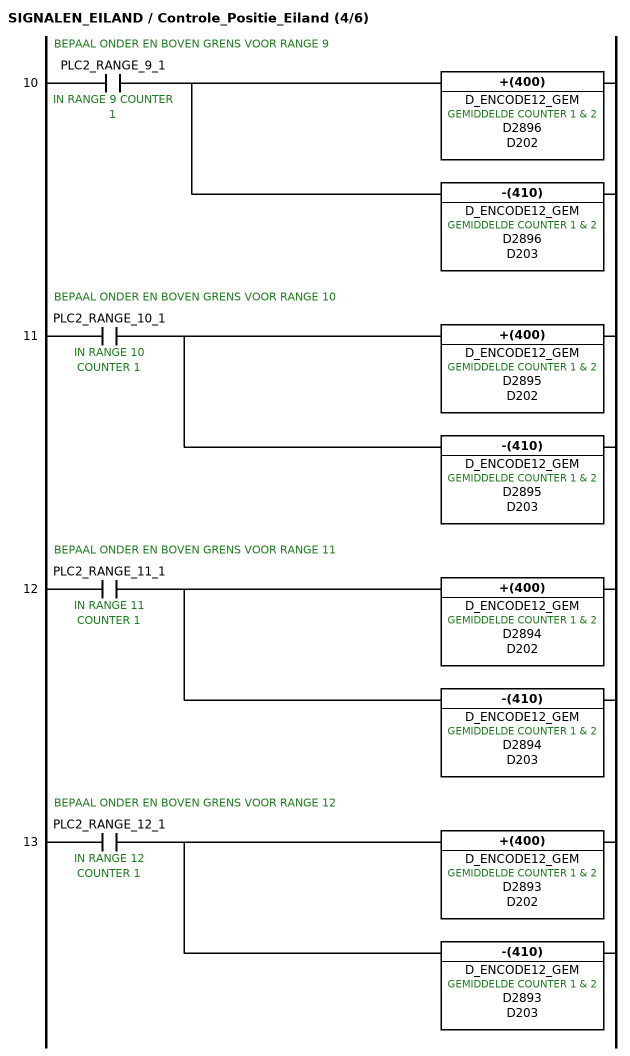
; [picture p397: SIGNALEN_EILAND / Controle_Positie_Eiland, rungs 10-13]
; rung 10: BEPAAL ONDER EN BOVEN GRENS VOOR RANGE 9
LD PLC2_RANGE_9_1  ; IN RANGE 9 COUNTER 1
+(400) D_ENCODE12_GEM D2896 D202  ; GEMIDDELDE COUNTER 1 & 2
-(410) D_ENCODE12_GEM D2896 D203  ; GEMIDDELDE COUNTER 1 & 2
; rung 11: BEPAAL ONDER EN BOVEN GRENS VOOR RANGE 10
LD PLC2_RANGE_10_1  ; IN RANGE 10 COUNTER 1
+(400) D_ENCODE12_GEM D2895 D202  ; GEMIDDELDE COUNTER 1 & 2
-(410) D_ENCODE12_GEM D2895 D203  ; GEMIDDELDE COUNTER 1 & 2
; rung 12: BEPAAL ONDER EN BOVEN GRENS VOOR RANGE 11
LD PLC2_RANGE_11_1  ; IN RANGE 11 COUNTER 1
+(400) D_ENCODE12_GEM D2894 D202  ; GEMIDDELDE COUNTER 1 & 2
-(410) D_ENCODE12_GEM D2894 D203  ; GEMIDDELDE COUNTER 1 & 2
; rung 13: BEPAAL ONDER EN BOVEN GRENS VOOR RANGE 12
LD PLC2_RANGE_12_1  ; IN RANGE 12 COUNTER 1
+(400) D_ENCODE12_GEM D2893 D202  ; GEMIDDELDE COUNTER 1 & 2
-(410) D_ENCODE12_GEM D2893 D203  ; GEMIDDELDE COUNTER 1 & 2

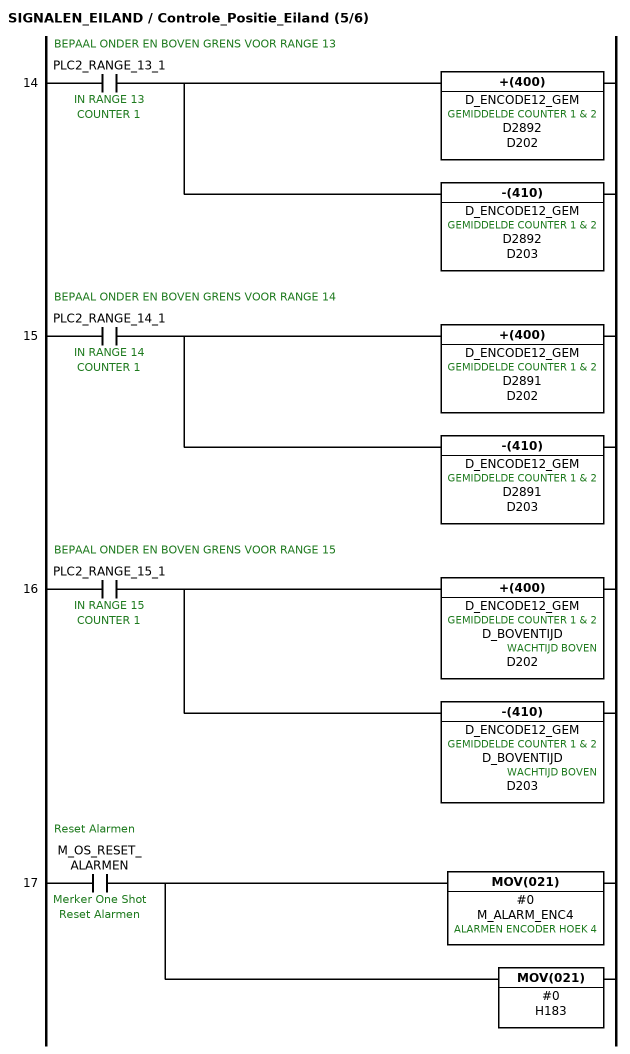
; rung 14: BEPAAL ONDER EN BOVEN GRENS VOOR RANGE 13
LD PLC2_RANGE_13_1  ; IN RANGE 13 COUNTER 1
+(400) D_ENCODE12_GEM D2892 D202  ; GEMIDDELDE COUNTER 1 & 2
-(410) D_ENCODE12_GEM D2892 D203  ; GEMIDDELDE COUNTER 1 & 2
; rung 15: BEPAAL ONDER EN BOVEN GRENS VOOR RANGE 14
LD PLC2_RANGE_14_1  ; IN RANGE 14 COUNTER 1
+(400) D_ENCODE12_GEM D2891 D202  ; GEMIDDELDE COUNTER 1 & 2
-(410) D_ENCODE12_GEM D2891 D203  ; GEMIDDELDE COUNTER 1 & 2
; rung 16: BEPAAL ONDER EN BOVEN GRENS VOOR RANGE 15
LD PLC2_RANGE_15_1  ; IN RANGE 15 COUNTER 1
+(400) D_ENCODE12_GEM D_BOVENTIJD D202  ; GEMIDDELDE COUNTER 1 & 2, WACHTIJD BOVEN
-(410) D_ENCODE12_GEM D_BOVENTIJD D203  ; GEMIDDELDE COUNTER 1 & 2, WACHTIJD BOVEN
; rung 17: Reset Alarmen
LD M_OS_RESET_ALARMEN  ; Merker One Shot Reset Alarmen
MOV(021) #0 M_ALARM_ENC4  ; ALARMEN ENCODER HOEK 4
MOV(021) #0 H183

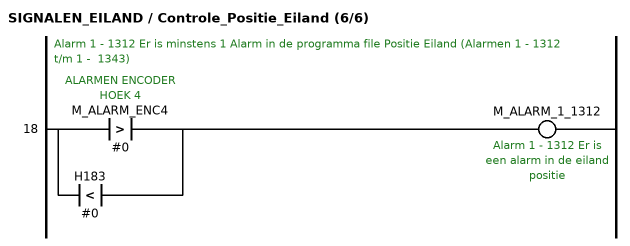
; rung 18: Alarm 1 - 1312 Er is minstens 1 Alarm in de programma file Positie Eiland (Alarmen 1 - 1312 t/m 1 -  1343)
LD>(320) M_ALARM_ENC4 #0  ; ALARMEN ENCODER HOEK 4
OR<(310) H183 #0
OUT M_ALARM_1_1312  ; Alarm 1 - 1312 Er is een alarm in de eiland positie

### Section Controle_Level_Switches_Eiland

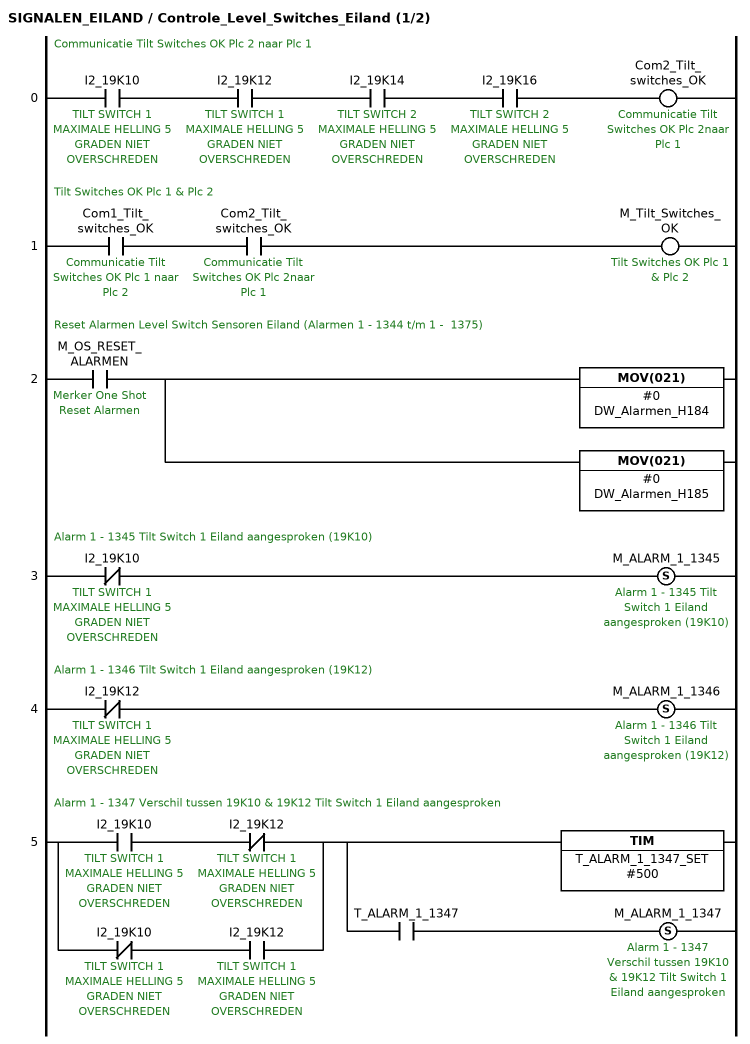
; rung 0: Communicatie Tilt Switches OK Plc 2 naar Plc 1
LD I2_19K10  ; TILT SWITCH 1 MAXIMALE HELLING 5 GRADEN NIET OVERSCHREDEN
AND I2_19K12  ; TILT SWITCH 1 MAXIMALE HELLING 5 GRADEN NIET OVERSCHREDEN
AND I2_19K14  ; TILT SWITCH 2 MAXIMALE HELLING 5 GRADEN NIET OVERSCHREDEN
AND I2_19K16  ; TILT SWITCH 2 MAXIMALE HELLING 5 GRADEN NIET OVERSCHREDEN
OUT Com2_Tilt_switches_OK  ; Communicatie Tilt Switches OK Plc 2naar Plc 1
; rung 1: Tilt Switches OK Plc 1 & Plc 2
LD Com1_Tilt_switches_OK  ; Communicatie Tilt Switches OK Plc 1 naar Plc 2
AND Com2_Tilt_switches_OK  ; Communicatie Tilt Switches OK Plc 2naar Plc 1
OUT M_Tilt_Switches_OK  ; Tilt Switches OK Plc 1 & Plc 2
; rung 2: Reset Alarmen Level Switch Sensoren Eiland (Alarmen 1 - 1344 t/m 1 -  1375)
LD M_OS_RESET_ALARMEN  ; Merker One Shot Reset Alarmen
MOV(021) #0 DW_Alarmen_H184
MOV(021) #0 DW_Alarmen_H185
; rung 3: Alarm 1 - 1345 Tilt Switch 1 Eiland aangesproken (19K10)
LDNOT I2_19K10  ; TILT SWITCH 1 MAXIMALE HELLING 5 GRADEN NIET OVERSCHREDEN
SET M_ALARM_1_1345  ; Alarm 1 - 1345 Tilt Switch 1 Eiland aangesproken (19K10)
; rung 4: Alarm 1 - 1346 Tilt Switch 1 Eiland aangesproken (19K12)
LDNOT I2_19K12  ; TILT SWITCH 1 MAXIMALE HELLING 5 GRADEN NIET OVERSCHREDEN
SET M_ALARM_1_1346  ; Alarm 1 - 1346 Tilt Switch 1 Eiland aangesproken (19K12)
; rung 5: Alarm 1 - 1347 Verschil tussen 19K10 & 19K12 Tilt Switch 1 Eiland aangesproken
LD I2_19K10  ; TILT SWITCH 1 MAXIMALE HELLING 5 GRADEN NIET OVERSCHREDEN
ANDNOT I2_19K12  ; TILT SWITCH 1 MAXIMALE HELLING 5 GRADEN NIET OVERSCHREDEN
LDNOT I2_19K10  ; TILT SWITCH 1 MAXIMALE HELLING 5 GRADEN NIET OVERSCHREDEN
AND I2_19K12  ; TILT SWITCH 1 MAXIMALE HELLING 5 GRADEN NIET OVERSCHREDEN
ORLD
TIM T_ALARM_1_1347_SET #500
AND T_ALARM_1_1347
SET M_ALARM_1_1347  ; Alarm 1 - 1347 Verschil tussen 19K10 & 19K12 Tilt Switch 1 Eiland aangesproken

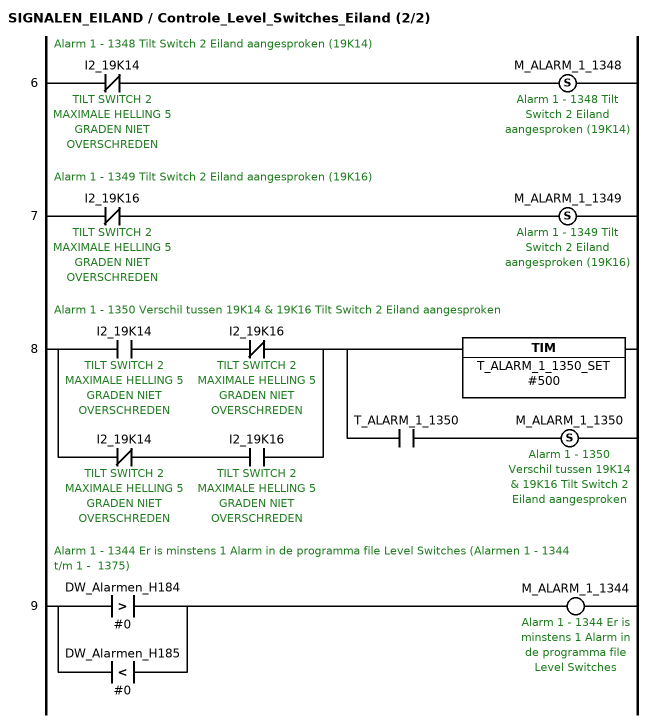
; rung 6: Alarm 1 - 1348 Tilt Switch 2 Eiland aangesproken (19K14)
LDNOT I2_19K14  ; TILT SWITCH 2 MAXIMALE HELLING 5 GRADEN NIET OVERSCHREDEN
SET M_ALARM_1_1348  ; Alarm 1 - 1348 Tilt Switch 2 Eiland aangesproken (19K14)
; rung 7: Alarm 1 - 1349 Tilt Switch 2 Eiland aangesproken (19K16)
LDNOT I2_19K16  ; TILT SWITCH 2 MAXIMALE HELLING 5 GRADEN NIET OVERSCHREDEN
SET M_ALARM_1_1349  ; Alarm 1 - 1349 Tilt Switch 2 Eiland aangesproken (19K16)
; rung 8: Alarm 1 - 1350 Verschil tussen 19K14 & 19K16 Tilt Switch 2 Eiland aangesproken
LD I2_19K14  ; TILT SWITCH 2 MAXIMALE HELLING 5 GRADEN NIET OVERSCHREDEN
ANDNOT I2_19K16  ; TILT SWITCH 2 MAXIMALE HELLING 5 GRADEN NIET OVERSCHREDEN
LDNOT I2_19K14  ; TILT SWITCH 2 MAXIMALE HELLING 5 GRADEN NIET OVERSCHREDEN
AND I2_19K16  ; TILT SWITCH 2 MAXIMALE HELLING 5 GRADEN NIET OVERSCHREDEN
ORLD
TIM T_ALARM_1_1350_SET #500
AND T_ALARM_1_1350
SET M_ALARM_1_1350  ; Alarm 1 - 1350 Verschil tussen 19K14 & 19K16 Tilt Switch 2 Eiland aangesproken
; rung 9: Alarm 1 - 1344 Er is minstens 1 Alarm in de programma file Level Switches (Alarmen 1 - 1344 t/m 1 -  1375)
LD>(320) DW_Alarmen_H184 #0
OR<(310) DW_Alarmen_H185 #0
OUT M_ALARM_1_1344  ; Alarm 1 - 1344 Er is minstens 1 Alarm in de programma file Level Switches

### Section Einde_Signalering_Eiland
; rung 0
END(001)

## Program BESTURING_EILAND (cyclic task 11)
Local symbols
Com1_Eiland_Rond_Geweest 3047.14 BOOL
Com1_Hydrauliek_Eiland_Inbedrijf 3045.15 BOOL
Com2_Eiland_Rond_Geweest 3347.14 BOOL
Com2_Hydrauliek_Eiland_Inbedrijf 3345.15 BOOL
M_ALARM_2_1515 H194.11 BOOL  ; Alarm 2 - 1515 Thermistor Fout Motor 2 Eiland (13R7 / 13U6 / 13K9)
M_Hoofdpomp_Hydrau_Eiland W220.03 BOOL  ; Start Hoofdpomp Hydrauliek Eiland

### Section Poortjes_Eiland

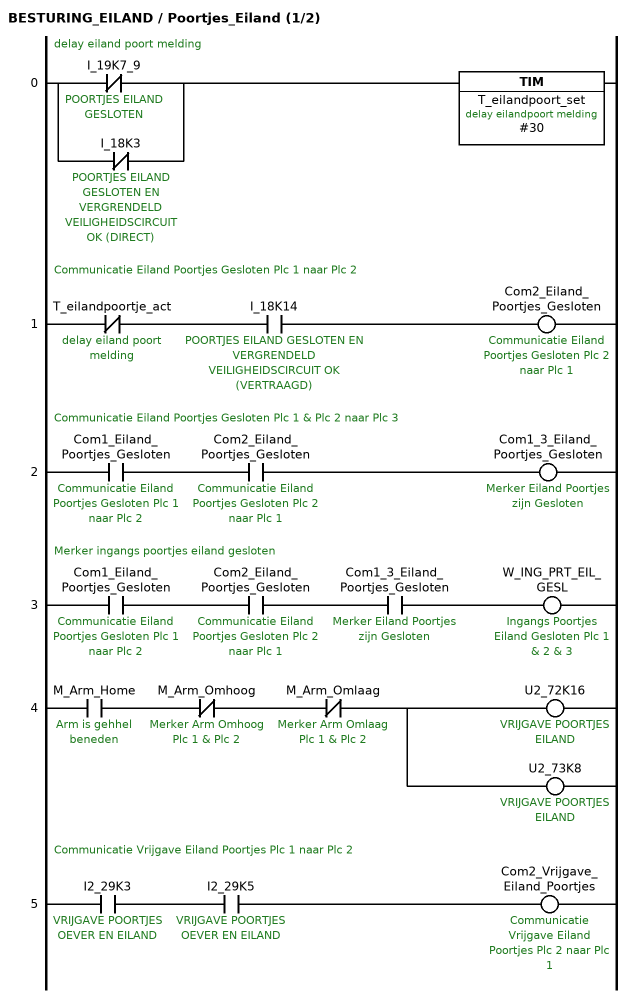
; rung 0: delay eiland poort melding
LDNOT I_19K7_9  ; POORTJES EILAND GESLOTEN
ORNOT I_18K3  ; POORTJES EILAND GESLOTEN EN VERGRENDELD VEILIGHEIDSCIRCUIT OK (DIRECT)
TIM T_eilandpoort_set #30  ; delay eilandpoort melding
; rung 1: Communicatie Eiland Poortjes Gesloten Plc 1 naar Plc 2
LDNOT T_eilandpoortje_act  ; delay eiland poort melding
AND I_18K14  ; POORTJES EILAND GESLOTEN EN VERGRENDELD VEILIGHEIDSCIRCUIT OK (VERTRAAGD)
OUT Com2_Eiland_Poortjes_Gesloten  ; Communicatie Eiland Poortjes Gesloten Plc 2 naar Plc 1
; rung 2: Communicatie Eiland Poortjes Gesloten Plc 1 & Plc 2 naar Plc 3
LD Com1_Eiland_Poortjes_Gesloten  ; Communicatie Eiland Poortjes Gesloten Plc 1 naar Plc 2
AND Com2_Eiland_Poortjes_Gesloten  ; Communicatie Eiland Poortjes Gesloten Plc 2 naar Plc 1
OUT Com1_3_Eiland_Poortjes_Gesloten  ; Merker Eiland Poortjes zijn Gesloten
; rung 3: Merker ingangs poortjes eiland gesloten
LD Com1_Eiland_Poortjes_Gesloten  ; Communicatie Eiland Poortjes Gesloten Plc 1 naar Plc 2
AND Com2_Eiland_Poortjes_Gesloten  ; Communicatie Eiland Poortjes Gesloten Plc 2 naar Plc 1
AND Com1_3_Eiland_Poortjes_Gesloten  ; Merker Eiland Poortjes zijn Gesloten
OUT W_ING_PRT_EIL_GESL  ; Ingangs Poortjes Eiland Gesloten Plc 1 & 2 & 3
; rung 4
LD M_Arm_Home  ; Arm is gehhel beneden
ANDNOT M_Arm_Omhoog  ; Merker Arm Omhoog Plc 1 & Plc 2
ANDNOT M_Arm_Omlaag  ; Merker Arm Omlaag Plc 1 & Plc 2
OUT U2_72K16  ; VRIJGAVE POORTJES EILAND
OUT U2_73K8  ; VRIJGAVE POORTJES EILAND
; rung 5: Communicatie Vrijgave Eiland Poortjes Plc 1 naar Plc 2
LD I2_29K3  ; VRIJGAVE POORTJES OEVER EN EILAND
AND I2_29K5  ; VRIJGAVE POORTJES OEVER EN EILAND
OUT Com2_Vrijgave_Eiland_Poortjes  ; Communicatie Vrijgave Eiland Poortjes Plc 2 naar Plc 1

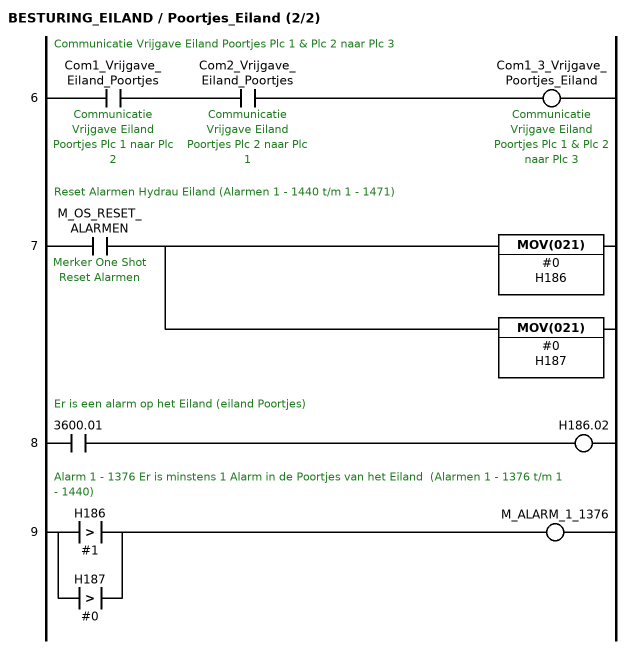
; rung 6: Communicatie Vrijgave Eiland Poortjes Plc 1 & Plc 2 naar Plc 3
LD Com1_Vrijgave_Eiland_Poortjes  ; Communicatie Vrijgave Eiland Poortjes Plc 1 naar Plc 2
AND Com2_Vrijgave_Eiland_Poortjes  ; Communicatie Vrijgave Eiland Poortjes Plc 2 naar Plc 1
OUT Com1_3_Vrijgave_Poortjes_Eiland  ; Communicatie Vrijgave Eiland Poortjes Plc 1 & Plc 2 naar Plc 3
; rung 7: Reset Alarmen Hydrau Eiland (Alarmen 1 - 1440 t/m 1 - 1471)
LD M_OS_RESET_ALARMEN  ; Merker One Shot Reset Alarmen
MOV(021) #0 H186
MOV(021) #0 H187
; rung 8: Er is een alarm op het Eiland (eiland Poortjes)
LD 3600.01
OUT H186.02
; rung 9: Alarm 1 - 1376 Er is minstens 1 Alarm in de Poortjes van het Eiland  (Alarmen 1 - 1376 t/m 1 - 1440)
LD>(320) H186 #1
OR>(320) H187 #0
OUT M_ALARM_1_1376

### Section Hydrauliek_Eiland

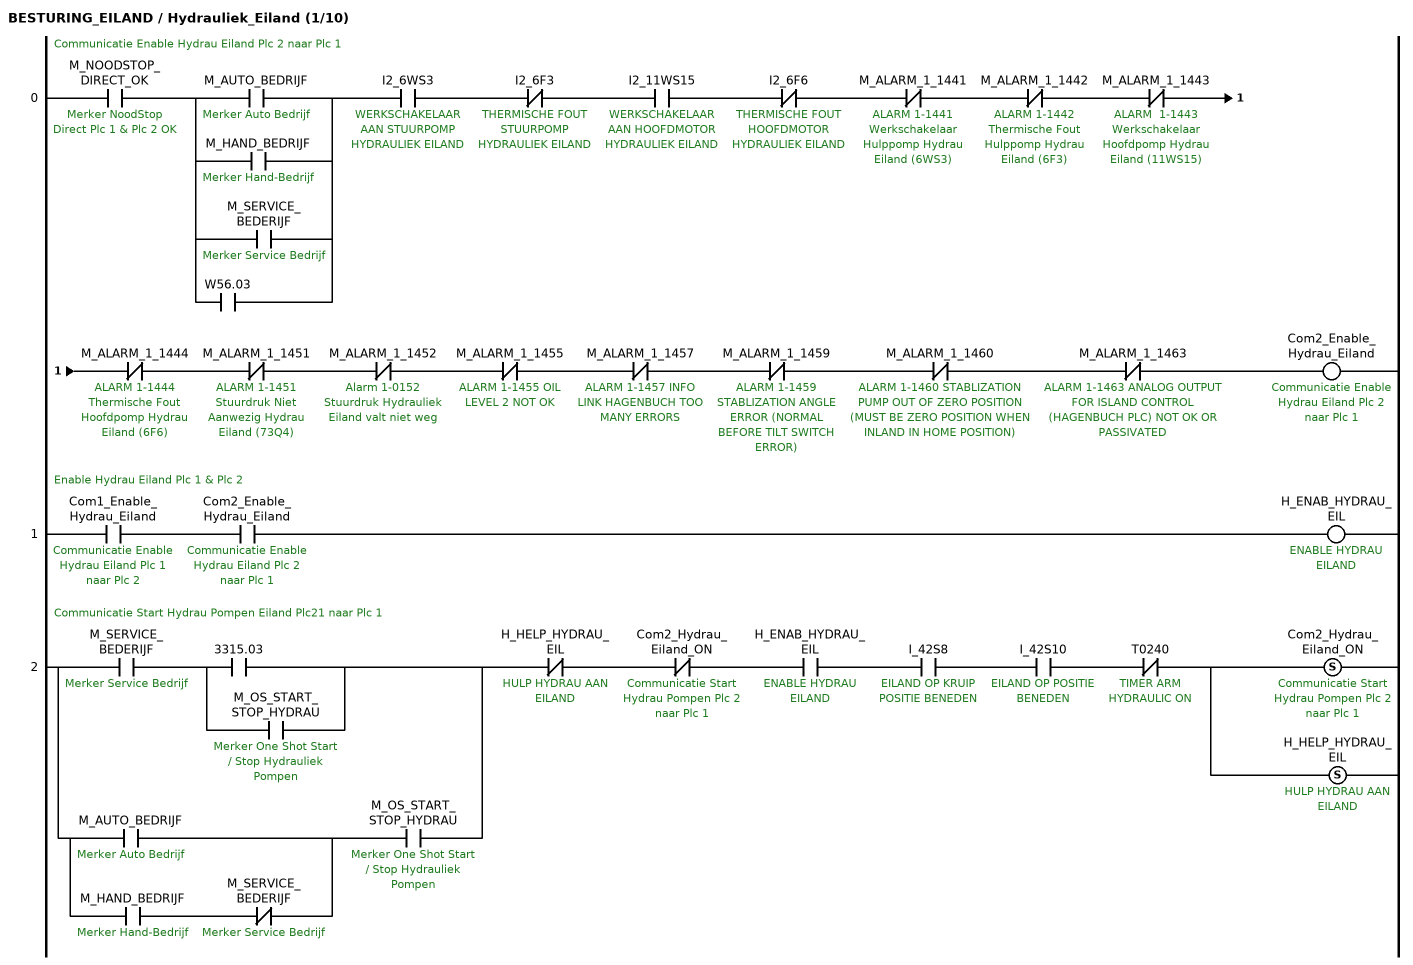
; rung 0: Communicatie Enable Hydrau Eiland Plc 2 naar Plc 1
LD M_NOODSTOP_DIRECT_OK  ; Merker NoodStop Direct Plc 1 & Plc 2 OK
LD M_AUTO_BEDRIJF  ; Merker Auto Bedrijf
OR M_HAND_BEDRIJF  ; Merker Hand-Bedrijf
OR M_SERVICE_BEDERIJF  ; Merker Service Bedrijf
OR W56.03
ANDLD
AND I2_6WS3  ; WERKSCHAKELAAR AAN STUURPOMP HYDRAULIEK EILAND
ANDNOT I2_6F3  ; THERMISCHE FOUT STUURPOMP HYDRAULIEK EILAND
AND I2_11WS15  ; WERKSCHAKELAAR AAN HOOFDMOTOR HYDRAULIEK EILAND
ANDNOT I2_6F6  ; THERMISCHE FOUT HOOFDMOTOR HYDRAULIEK EILAND
ANDNOT M_ALARM_1_1441  ; ALARM 1-1441 Werkschakelaar Hulppomp Hydrau Eiland (6WS3)
ANDNOT M_ALARM_1_1442  ; ALARM 1-1442 Thermische Fout Hulppomp Hydrau Eiland (6F3)
ANDNOT M_ALARM_1_1443  ; ALARM  1-1443 Werkschakelaar Hoofdpomp Hydrau Eiland (11WS15)
ANDNOT M_ALARM_1_1444  ; ALARM 1-1444 Thermische Fout Hoofdpomp Hydrau Eiland (6F6)
ANDNOT M_ALARM_1_1451  ; ALARM 1-1451 Stuurdruk Niet Aanwezig Hydrau Eiland (73Q4)
ANDNOT M_ALARM_1_1452  ; Alarm 1-0152 Stuurdruk Hydrauliek Eiland valt niet weg
ANDNOT M_ALARM_1_1455  ; ALARM 1-1455 OIL LEVEL 2 NOT OK
ANDNOT M_ALARM_1_1457  ; ALARM 1-1457 INFO LINK HAGENBUCH TOO MANY ERRORS
ANDNOT M_ALARM_1_1459  ; ALARM 1-1459 STABLIZATION ANGLE ERROR (NORMAL BEFORE TILT SWITCH ERROR)
ANDNOT M_ALARM_1_1460  ; ALARM 1-1460 STABLIZATION PUMP OUT OF ZERO POSITION (MUST BE ZERO POSITION WHEN INLAND IN HOME POSITION)
ANDNOT M_ALARM_1_1463  ; ALARM 1-1463 ANALOG OUTPUT FOR ISLAND CONTROL (HAGENBUCH PLC) NOT OK OR PASSIVATED
OUT Com2_Enable_Hydrau_Eiland  ; Communicatie Enable Hydrau Eiland Plc 2 naar Plc 1
; rung 1: Enable Hydrau Eiland Plc 1 & Plc 2
LD Com1_Enable_Hydrau_Eiland  ; Communicatie Enable Hydrau Eiland Plc 1 naar Plc 2
AND Com2_Enable_Hydrau_Eiland  ; Communicatie Enable Hydrau Eiland Plc 2 naar Plc 1
OUT H_ENAB_HYDRAU_EIL  ; ENABLE HYDRAU EILAND
; rung 2: Communicatie Start Hydrau Pompen Eiland Plc21 naar Plc 1
LD M_SERVICE_BEDERIJF  ; Merker Service Bedrijf
LD 3315.03
OR M_OS_START_STOP_HYDRAU  ; Merker One Shot Start / Stop Hydrauliek Pompen
ANDLD
LD M_AUTO_BEDRIJF  ; Merker Auto Bedrijf
LD M_HAND_BEDRIJF  ; Merker Hand-Bedrijf
ANDNOT M_SERVICE_BEDERIJF  ; Merker Service Bedrijf
ORLD
AND M_OS_START_STOP_HYDRAU  ; Merker One Shot Start / Stop Hydrauliek Pompen
ORLD
ANDNOT H_HELP_HYDRAU_EIL  ; HULP HYDRAU AAN EILAND
ANDNOT Com2_Hydrau_Eiland_ON  ; Communicatie Start Hydrau Pompen Plc 2 naar Plc 1
AND H_ENAB_HYDRAU_EIL  ; ENABLE HYDRAU EILAND
AND I_42S8  ; EILAND OP KRUIP POSITIE BENEDEN
AND I_42S10  ; EILAND OP POSITIE BENEDEN
ANDNOT T0240  ; TIMER ARM HYDRAULIC ON
SET Com2_Hydrau_Eiland_ON  ; Communicatie Start Hydrau Pompen Plc 2 naar Plc 1
SET H_HELP_HYDRAU_EIL  ; HULP HYDRAU AAN EILAND

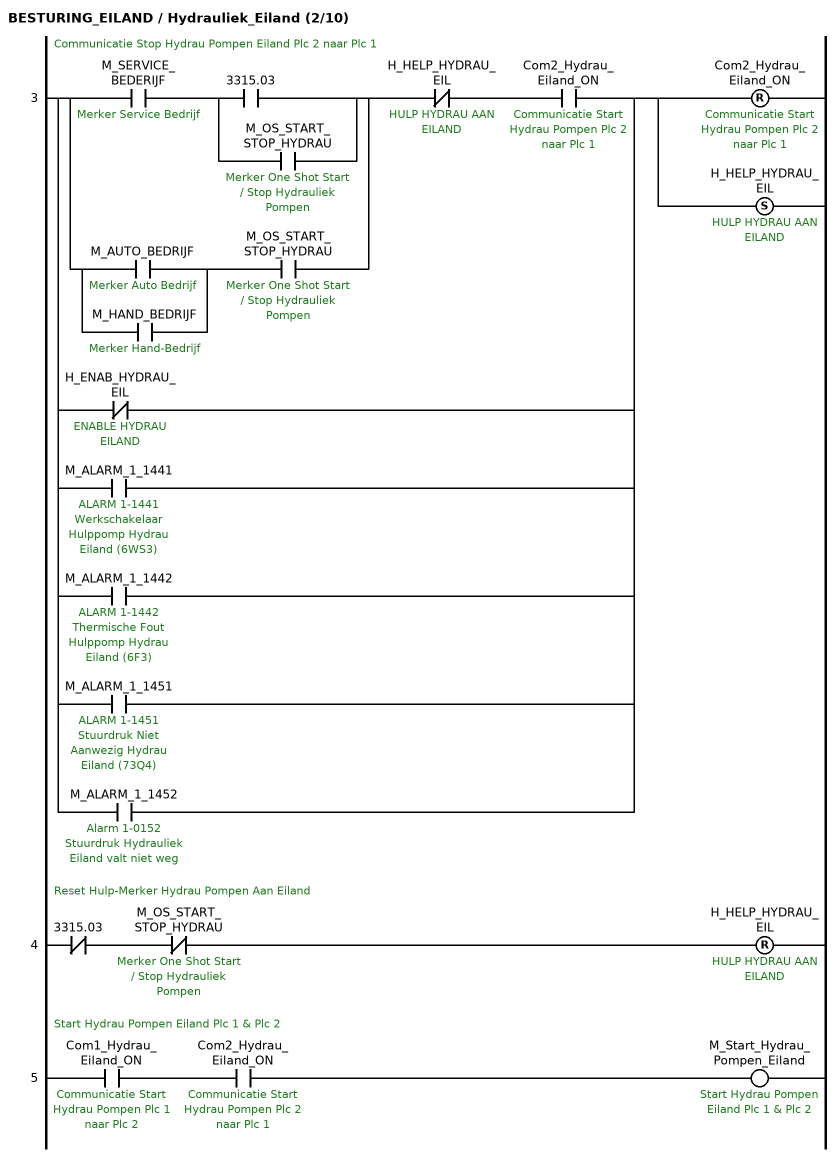
; rung 3: Communicatie Stop Hydrau Pompen Eiland Plc 2 naar Plc 1
LD M_SERVICE_BEDERIJF  ; Merker Service Bedrijf
LD 3315.03
OR M_OS_START_STOP_HYDRAU  ; Merker One Shot Start / Stop Hydrauliek Pompen
ANDLD
LD M_AUTO_BEDRIJF  ; Merker Auto Bedrijf
OR M_HAND_BEDRIJF  ; Merker Hand-Bedrijf
AND M_OS_START_STOP_HYDRAU  ; Merker One Shot Start / Stop Hydrauliek Pompen
ORLD
ANDNOT H_HELP_HYDRAU_EIL  ; HULP HYDRAU AAN EILAND
AND Com2_Hydrau_Eiland_ON  ; Communicatie Start Hydrau Pompen Plc 2 naar Plc 1
ORNOT H_ENAB_HYDRAU_EIL  ; ENABLE HYDRAU EILAND
OR M_ALARM_1_1441  ; ALARM 1-1441 Werkschakelaar Hulppomp Hydrau Eiland (6WS3)
OR M_ALARM_1_1442  ; ALARM 1-1442 Thermische Fout Hulppomp Hydrau Eiland (6F3)
OR M_ALARM_1_1451  ; ALARM 1-1451 Stuurdruk Niet Aanwezig Hydrau Eiland (73Q4)
OR M_ALARM_1_1452  ; Alarm 1-0152 Stuurdruk Hydrauliek Eiland valt niet weg
RSET Com2_Hydrau_Eiland_ON  ; Communicatie Start Hydrau Pompen Plc 2 naar Plc 1
SET H_HELP_HYDRAU_EIL  ; HULP HYDRAU AAN EILAND
; rung 4: Reset Hulp-Merker Hydrau Pompen Aan Eiland
LDNOT 3315.03
ANDNOT M_OS_START_STOP_HYDRAU  ; Merker One Shot Start / Stop Hydrauliek Pompen
RSET H_HELP_HYDRAU_EIL  ; HULP HYDRAU AAN EILAND
; rung 5: Start Hydrau Pompen Eiland Plc 1 & Plc 2
LD Com1_Hydrau_Eiland_ON  ; Communicatie Start Hydrau Pompen Plc 1 naar Plc 2
AND Com2_Hydrau_Eiland_ON  ; Communicatie Start Hydrau Pompen Plc 2 naar Plc 1
OUT M_Start_Hydrau_Pompen_Eiland  ; Start Hydrau Pompen Eiland Plc 1 & Plc 2

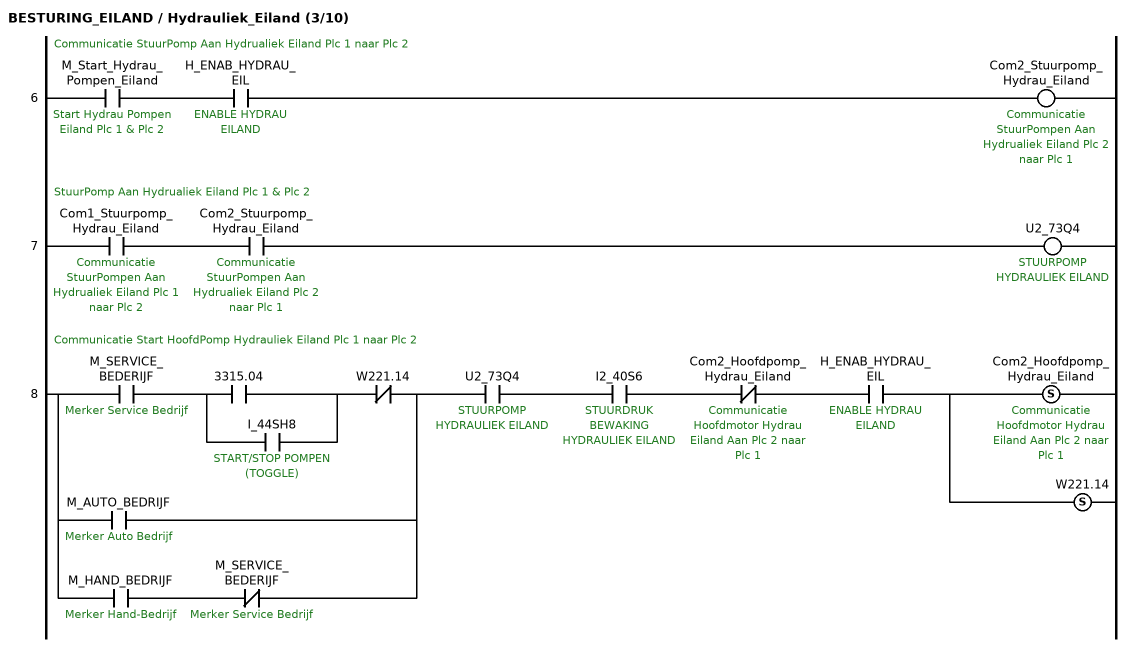
; rung 6: Communicatie StuurPomp Aan Hydrualiek Eiland Plc 1 naar Plc 2
LD M_Start_Hydrau_Pompen_Eiland  ; Start Hydrau Pompen Eiland Plc 1 & Plc 2
AND H_ENAB_HYDRAU_EIL  ; ENABLE HYDRAU EILAND
OUT Com2_Stuurpomp_Hydrau_Eiland  ; Communicatie StuurPompen Aan Hydrualiek Eiland Plc 2 naar Plc 1
; rung 7: StuurPomp Aan Hydrualiek Eiland Plc 1 & Plc 2
LD Com1_Stuurpomp_Hydrau_Eiland  ; Communicatie StuurPompen Aan Hydrualiek Eiland Plc 1 naar Plc 2
AND Com2_Stuurpomp_Hydrau_Eiland  ; Communicatie StuurPompen Aan Hydrualiek Eiland Plc 2 naar Plc 1
OUT U2_73Q4  ; STUURPOMP HYDRAULIEK EILAND
; rung 8: Communicatie Start HoofdPomp Hydrauliek Eiland Plc 1 naar Plc 2
LD M_SERVICE_BEDERIJF  ; Merker Service Bedrijf
LD 3315.04
OR I_44SH8  ; START/STOP POMPEN (TOGGLE)
ANDLD
ANDNOT W221.14
OR M_AUTO_BEDRIJF  ; Merker Auto Bedrijf
LD M_HAND_BEDRIJF  ; Merker Hand-Bedrijf
ANDNOT M_SERVICE_BEDERIJF  ; Merker Service Bedrijf
ORLD
AND U2_73Q4  ; STUURPOMP HYDRAULIEK EILAND
AND I2_40S6  ; STUURDRUK BEWAKING HYDRAULIEK EILAND
ANDNOT Com2_Hoofdpomp_Hydrau_Eiland  ; Communicatie Hoofdmotor Hydrau Eiland Aan Plc 2 naar Plc 1
AND H_ENAB_HYDRAU_EIL  ; ENABLE HYDRAU EILAND
SET Com2_Hoofdpomp_Hydrau_Eiland  ; Communicatie Hoofdmotor Hydrau Eiland Aan Plc 2 naar Plc 1
SET W221.14

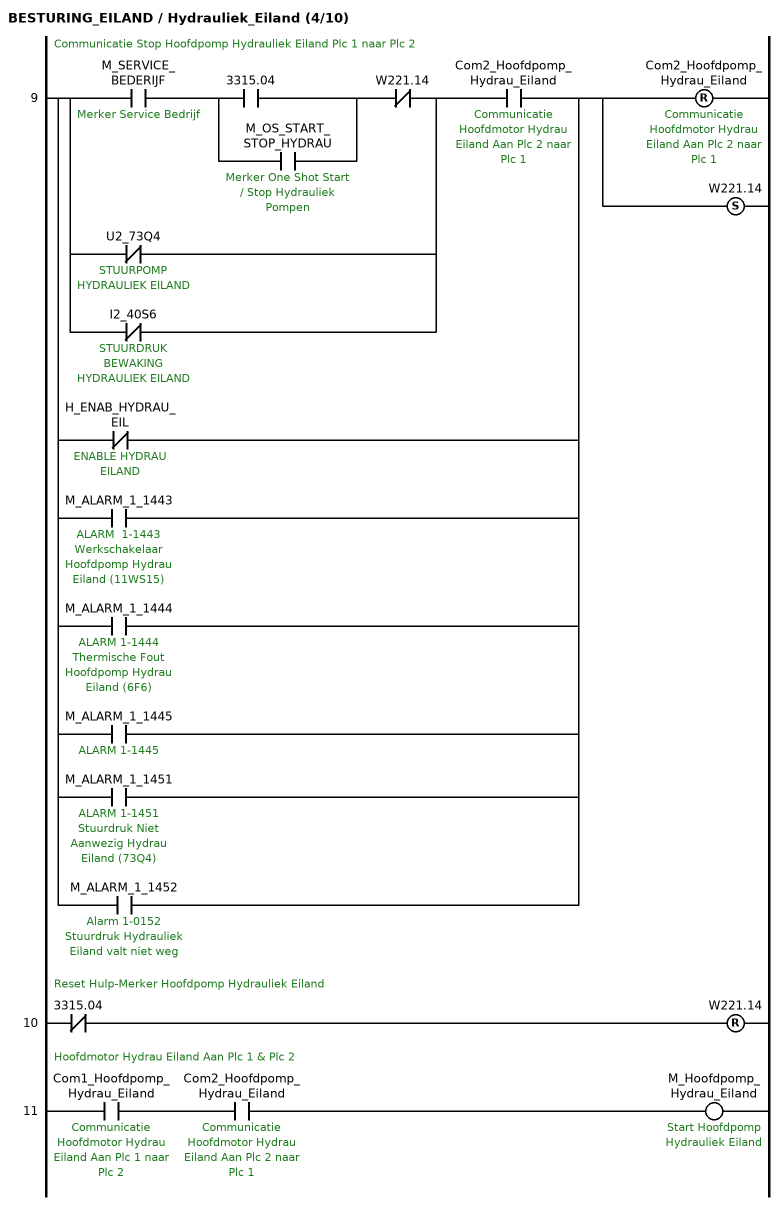
; rung 9: Communicatie Stop Hoofdpomp Hydrauliek Eiland Plc 1 naar Plc 2
LD M_SERVICE_BEDERIJF  ; Merker Service Bedrijf
LD 3315.04
OR M_OS_START_STOP_HYDRAU  ; Merker One Shot Start / Stop Hydrauliek Pompen
ANDLD
ANDNOT W221.14
ORNOT U2_73Q4  ; STUURPOMP HYDRAULIEK EILAND
ORNOT I2_40S6  ; STUURDRUK BEWAKING HYDRAULIEK EILAND
AND Com2_Hoofdpomp_Hydrau_Eiland  ; Communicatie Hoofdmotor Hydrau Eiland Aan Plc 2 naar Plc 1
ORNOT H_ENAB_HYDRAU_EIL  ; ENABLE HYDRAU EILAND
OR M_ALARM_1_1443  ; ALARM  1-1443 Werkschakelaar Hoofdpomp Hydrau Eiland (11WS15)
OR M_ALARM_1_1444  ; ALARM 1-1444 Thermische Fout Hoofdpomp Hydrau Eiland (6F6)
OR M_ALARM_1_1445  ; ALARM 1-1445
OR M_ALARM_1_1451  ; ALARM 1-1451 Stuurdruk Niet Aanwezig Hydrau Eiland (73Q4)
OR M_ALARM_1_1452  ; Alarm 1-0152 Stuurdruk Hydrauliek Eiland valt niet weg
RSET Com2_Hoofdpomp_Hydrau_Eiland  ; Communicatie Hoofdmotor Hydrau Eiland Aan Plc 2 naar Plc 1
SET W221.14
; rung 10: Reset Hulp-Merker Hoofdpomp Hydrauliek Eiland
LDNOT 3315.04
RSET W221.14
; rung 11: Hoofdmotor Hydrau Eiland Aan Plc 1 & Plc 2
LD Com1_Hoofdpomp_Hydrau_Eiland  ; Communicatie Hoofdmotor Hydrau Eiland Aan Plc 1 naar Plc 2
AND Com2_Hoofdpomp_Hydrau_Eiland  ; Communicatie Hoofdmotor Hydrau Eiland Aan Plc 2 naar Plc 1
OUT M_Hoofdpomp_Hydrau_Eiland  ; Start Hoofdpomp Hydrauliek Eiland

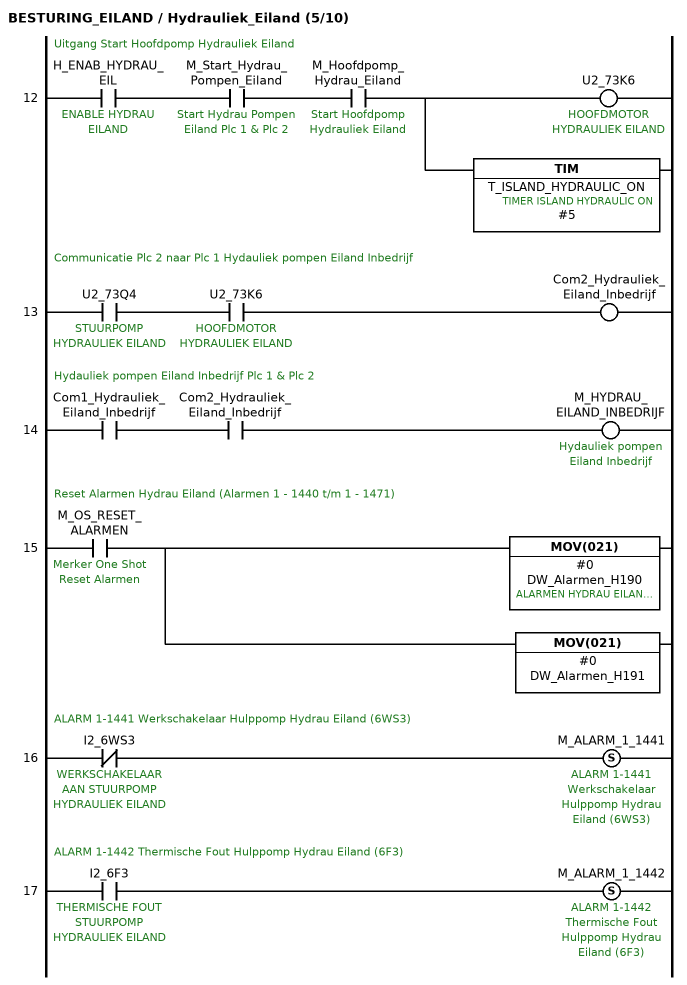
; rung 12: Uitgang Start Hoofdpomp Hydrauliek Eiland
LD H_ENAB_HYDRAU_EIL  ; ENABLE HYDRAU EILAND
AND M_Start_Hydrau_Pompen_Eiland  ; Start Hydrau Pompen Eiland Plc 1 & Plc 2
AND M_Hoofdpomp_Hydrau_Eiland  ; Start Hoofdpomp Hydrauliek Eiland
OUT U2_73K6  ; HOOFDMOTOR HYDRAULIEK EILAND
TIM T_ISLAND_HYDRAULIC_ON #5  ; TIMER ISLAND HYDRAULIC ON
; rung 13: Communicatie Plc 2 naar Plc 1 Hydauliek pompen Eiland Inbedrijf
LD U2_73Q4  ; STUURPOMP HYDRAULIEK EILAND
AND U2_73K6  ; HOOFDMOTOR HYDRAULIEK EILAND
OUT Com2_Hydrauliek_Eiland_Inbedrijf
; rung 14: Hydauliek pompen Eiland Inbedrijf Plc 1 & Plc 2
LD Com1_Hydrauliek_Eiland_Inbedrijf
AND Com2_Hydrauliek_Eiland_Inbedrijf
OUT M_HYDRAU_EILAND_INBEDRIJF  ; Hydauliek pompen Eiland Inbedrijf
; rung 15: Reset Alarmen Hydrau Eiland (Alarmen 1 - 1440 t/m 1 - 1471)
LD M_OS_RESET_ALARMEN  ; Merker One Shot Reset Alarmen
MOV(021) #0 DW_Alarmen_H190  ; ALARMEN HYDRAU EILAND 1440-1455
MOV(021) #0 DW_Alarmen_H191
; rung 16: ALARM 1-1441 Werkschakelaar Hulppomp Hydrau Eiland (6WS3)
LDNOT I2_6WS3  ; WERKSCHAKELAAR AAN STUURPOMP HYDRAULIEK EILAND
SET M_ALARM_1_1441  ; ALARM 1-1441 Werkschakelaar Hulppomp Hydrau Eiland (6WS3)
; rung 17: ALARM 1-1442 Thermische Fout Hulppomp Hydrau Eiland (6F3)
LD I2_6F3  ; THERMISCHE FOUT STUURPOMP HYDRAULIEK EILAND
SET M_ALARM_1_1442  ; ALARM 1-1442 Thermische Fout Hulppomp Hydrau Eiland (6F3)

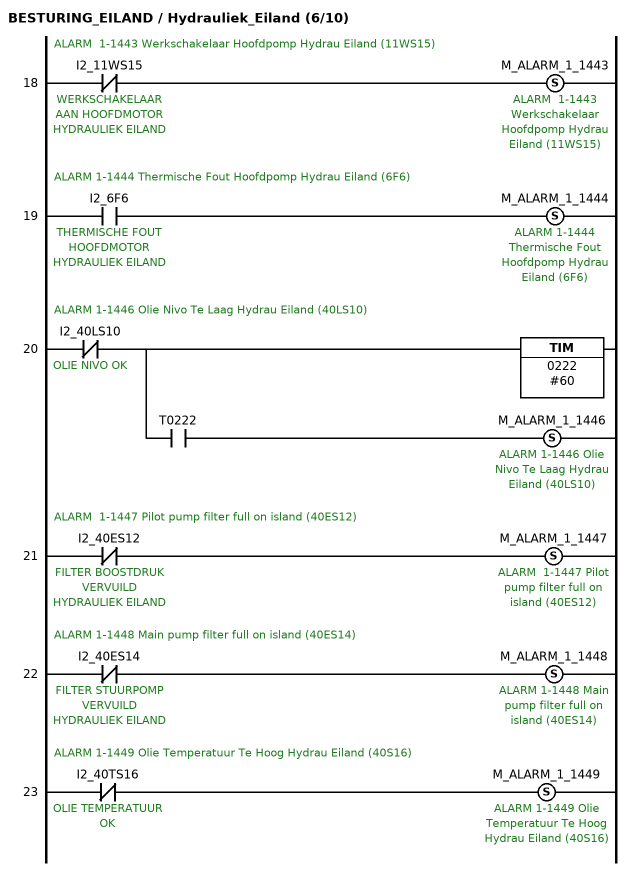
; rung 18: ALARM  1-1443 Werkschakelaar Hoofdpomp Hydrau Eiland (11WS15)
LDNOT I2_11WS15  ; WERKSCHAKELAAR AAN HOOFDMOTOR HYDRAULIEK EILAND
SET M_ALARM_1_1443  ; ALARM  1-1443 Werkschakelaar Hoofdpomp Hydrau Eiland (11WS15)
; rung 19: ALARM 1-1444 Thermische Fout Hoofdpomp Hydrau Eiland (6F6)
LD I2_6F6  ; THERMISCHE FOUT HOOFDMOTOR HYDRAULIEK EILAND
SET M_ALARM_1_1444  ; ALARM 1-1444 Thermische Fout Hoofdpomp Hydrau Eiland (6F6)
; rung 20: ALARM 1-1446 Olie Nivo Te Laag Hydrau Eiland (40LS10)
LDNOT I2_40LS10  ; OLIE NIVO OK
TIM 0222 #60
AND T0222
SET M_ALARM_1_1446  ; ALARM 1-1446 Olie Nivo Te Laag Hydrau Eiland (40LS10)
; rung 21: ALARM  1-1447 Pilot pump filter full on island (40ES12)
LDNOT I2_40ES12  ; FILTER BOOSTDRUK VERVUILD HYDRAULIEK EILAND
SET M_ALARM_1_1447  ; ALARM  1-1447 Pilot pump filter full on island (40ES12)
; rung 22: ALARM 1-1448 Main pump filter full on island (40ES14)
LDNOT I2_40ES14  ; FILTER STUURPOMP VERVUILD HYDRAULIEK EILAND
SET M_ALARM_1_1448  ; ALARM 1-1448 Main pump filter full on island (40ES14)
; rung 23: ALARM 1-1449 Olie Temperatuur Te Hoog Hydrau Eiland (40S16)
LDNOT I2_40TS16  ; OLIE TEMPERATUUR OK
SET M_ALARM_1_1449  ; ALARM 1-1449 Olie Temperatuur Te Hoog Hydrau Eiland (40S16)

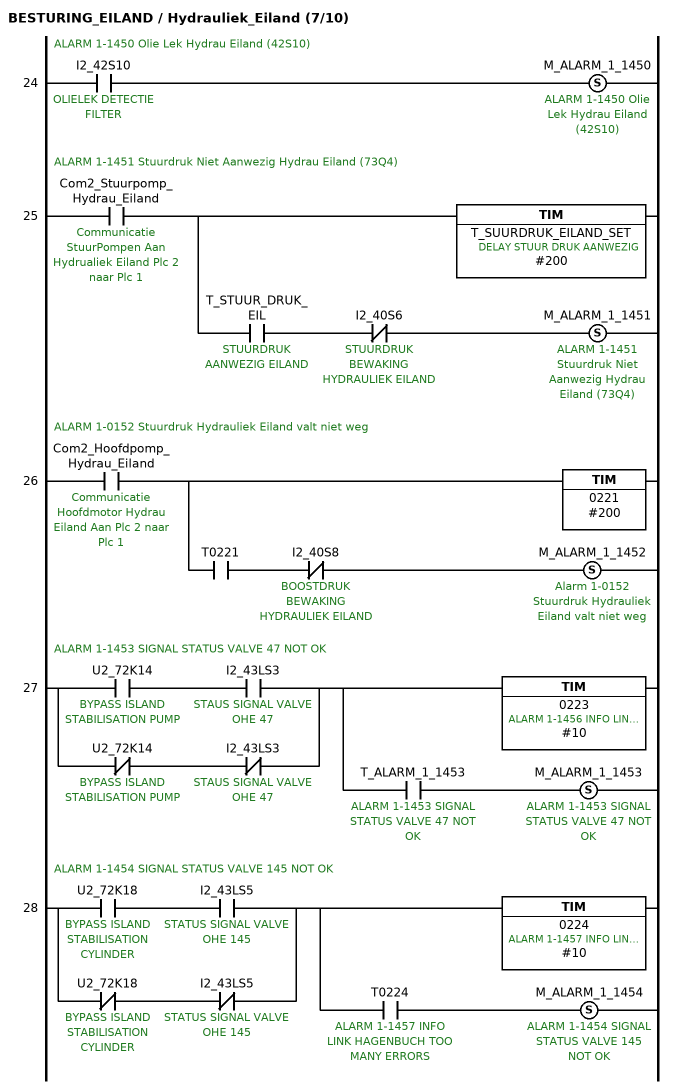
; rung 24: ALARM 1-1450 Olie Lek Hydrau Eiland (42S10)
LD I2_42S10  ; OLIELEK DETECTIE FILTER
SET M_ALARM_1_1450  ; ALARM 1-1450 Olie Lek Hydrau Eiland (42S10)
; rung 25: ALARM 1-1451 Stuurdruk Niet Aanwezig Hydrau Eiland (73Q4)
LD Com2_Stuurpomp_Hydrau_Eiland  ; Communicatie StuurPompen Aan Hydrualiek Eiland Plc 2 naar Plc 1
TIM T_SUURDRUK_EILAND_SET #200  ; DELAY STUUR DRUK AANWEZIG
AND T_STUUR_DRUK_EIL  ; STUURDRUK AANWEZIG EILAND
ANDNOT I2_40S6  ; STUURDRUK BEWAKING HYDRAULIEK EILAND
SET M_ALARM_1_1451  ; ALARM 1-1451 Stuurdruk Niet Aanwezig Hydrau Eiland (73Q4)
; rung 26: ALARM 1-0152 Stuurdruk Hydrauliek Eiland valt niet weg
LD Com2_Hoofdpomp_Hydrau_Eiland  ; Communicatie Hoofdmotor Hydrau Eiland Aan Plc 2 naar Plc 1
TIM 0221 #200
AND T0221
ANDNOT I2_40S8  ; BOOSTDRUK BEWAKING HYDRAULIEK EILAND
SET M_ALARM_1_1452  ; Alarm 1-0152 Stuurdruk Hydrauliek Eiland valt niet weg
; rung 27: ALARM 1-1453 SIGNAL STATUS VALVE 47 NOT OK
LD U2_72K14  ; BYPASS ISLAND STABILISATION PUMP
AND I2_43LS3  ; STAUS SIGNAL VALVE OHE 47
LDNOT U2_72K14  ; BYPASS ISLAND STABILISATION PUMP
ANDNOT I2_43LS3  ; STAUS SIGNAL VALVE OHE 47
ORLD
TIM 0223 #10  ; ALARM 1-1456 INFO LINK HAGENBUCH (FIBRE OPTIK) NOT AVAILABLE
AND T_ALARM_1_1453  ; ALARM 1-1453 SIGNAL STATUS VALVE 47 NOT OK
SET M_ALARM_1_1453  ; ALARM 1-1453 SIGNAL STATUS VALVE 47 NOT OK
; rung 28: ALARM 1-1454 SIGNAL STATUS VALVE 145 NOT OK
LD U2_72K18  ; BYPASS ISLAND STABILISATION CYLINDER
AND I2_43LS5  ; STATUS SIGNAL VALVE OHE 145
LDNOT U2_72K18  ; BYPASS ISLAND STABILISATION CYLINDER
ANDNOT I2_43LS5  ; STATUS SIGNAL VALVE OHE 145
ORLD
TIM 0224 #10  ; ALARM 1-1457 INFO LINK HAGENBUCH TOO MANY ERRORS
AND T0224  ; ALARM 1-1457 INFO LINK HAGENBUCH TOO MANY ERRORS
SET M_ALARM_1_1454  ; ALARM 1-1454 SIGNAL STATUS VALVE 145 NOT OK

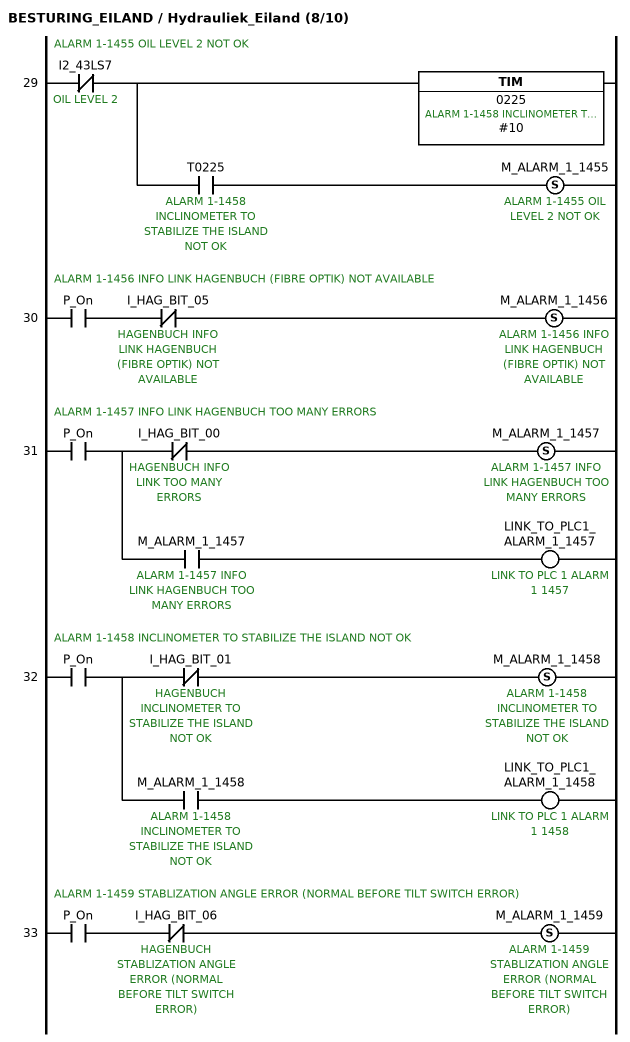
; rung 29: ALARM 1-1455 OIL LEVEL 2 NOT OK
LDNOT I2_43LS7  ; OIL LEVEL 2
TIM 0225 #10  ; ALARM 1-1458 INCLINOMETER TO STABILIZE THE ISLAND NOT OK
AND T0225  ; ALARM 1-1458 INCLINOMETER TO STABILIZE THE ISLAND NOT OK
SET M_ALARM_1_1455  ; ALARM 1-1455 OIL LEVEL 2 NOT OK
; rung 30: ALARM 1-1456 INFO LINK HAGENBUCH (FIBRE OPTIK) NOT AVAILABLE
LD P_On
ANDNOT I_HAG_BIT_05  ; HAGENBUCH INFO LINK HAGENBUCH (FIBRE OPTIK) NOT AVAILABLE
SET M_ALARM_1_1456  ; ALARM 1-1456 INFO LINK HAGENBUCH (FIBRE OPTIK) NOT AVAILABLE
; rung 31: ALARM 1-1457 INFO LINK HAGENBUCH TOO MANY ERRORS
LD P_On
OUT TR0
ANDNOT I_HAG_BIT_00  ; HAGENBUCH INFO LINK TOO MANY ERRORS
SET M_ALARM_1_1457  ; ALARM 1-1457 INFO LINK HAGENBUCH TOO MANY ERRORS
LD TR0
AND M_ALARM_1_1457  ; ALARM 1-1457 INFO LINK HAGENBUCH TOO MANY ERRORS
OUT LINK_TO_PLC1_ALARM_1_1457  ; LINK TO PLC 1 ALARM 1 1457
; rung 32: ALARM 1-1458 INCLINOMETER TO STABILIZE THE ISLAND NOT OK
LD P_On
OUT TR0
ANDNOT I_HAG_BIT_01  ; HAGENBUCH INCLINOMETER TO STABILIZE THE ISLAND NOT OK
SET M_ALARM_1_1458  ; ALARM 1-1458 INCLINOMETER TO STABILIZE THE ISLAND NOT OK
LD TR0
AND M_ALARM_1_1458  ; ALARM 1-1458 INCLINOMETER TO STABILIZE THE ISLAND NOT OK
OUT LINK_TO_PLC1_ALARM_1_1458  ; LINK TO PLC 1 ALARM 1 1458
; rung 33: ALARM 1-1459 STABLIZATION ANGLE ERROR (NORMAL BEFORE TILT SWITCH ERROR)
LD P_On
ANDNOT I_HAG_BIT_06  ; HAGENBUCH STABLIZATION ANGLE ERROR (NORMAL BEFORE TILT SWITCH ERROR)
SET M_ALARM_1_1459  ; ALARM 1-1459 STABLIZATION ANGLE ERROR (NORMAL BEFORE TILT SWITCH ERROR)

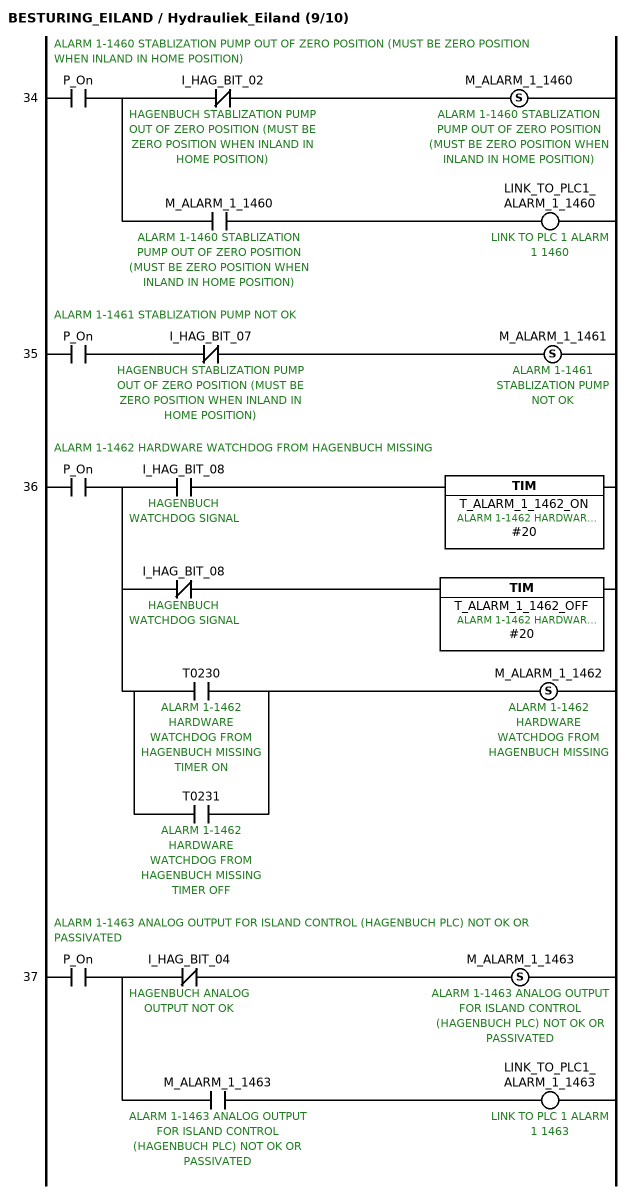
; rung 34: ALARM 1-1460 STABLIZATION PUMP OUT OF ZERO POSITION (MUST BE ZERO POSITION WHEN INLAND IN HOME POSITION)
LD P_On
OUT TR0
ANDNOT I_HAG_BIT_02  ; HAGENBUCH STABLIZATION PUMP OUT OF ZERO POSITION (MUST BE ZERO POSITION WHEN INLAND IN HOME POSITION)
SET M_ALARM_1_1460  ; ALARM 1-1460 STABLIZATION PUMP OUT OF ZERO POSITION (MUST BE ZERO POSITION WHEN INLAND IN HOME POSITION)
LD TR0
AND M_ALARM_1_1460  ; ALARM 1-1460 STABLIZATION PUMP OUT OF ZERO POSITION (MUST BE ZERO POSITION WHEN INLAND IN HOME POSITION)
OUT LINK_TO_PLC1_ALARM_1_1460  ; LINK TO PLC 1 ALARM 1 1460
; rung 35: ALARM 1-1461 STABLIZATION PUMP NOT OK
LD P_On
ANDNOT I_HAG_BIT_07  ; HAGENBUCH STABLIZATION PUMP OUT OF ZERO POSITION (MUST BE ZERO POSITION WHEN INLAND IN HOME POSITION)
SET M_ALARM_1_1461  ; ALARM 1-1461 STABLIZATION PUMP NOT OK
; rung 36: ALARM 1-1462 HARDWARE WATCHDOG FROM HAGENBUCH MISSING
LD P_On
OUT TR0
AND I_HAG_BIT_08  ; HAGENBUCH WATCHDOG SIGNAL
TIM T_ALARM_1_1462_ON #20  ; ALARM 1-1462 HARDWARE WATCHDOG FROM HAGENBUCH MISSING TIMER ON
LD TR0
ANDNOT I_HAG_BIT_08  ; HAGENBUCH WATCHDOG SIGNAL
TIM T_ALARM_1_1462_OFF #20  ; ALARM 1-1462 HARDWARE WATCHDOG FROM HAGENBUCH MISSING TIMER OFF
LD TR0
LD T0230  ; ALARM 1-1462 HARDWARE WATCHDOG FROM HAGENBUCH MISSING TIMER ON
OR T0231  ; ALARM 1-1462 HARDWARE WATCHDOG FROM HAGENBUCH MISSING TIMER OFF
ANDLD
SET M_ALARM_1_1462  ; ALARM 1-1462 HARDWARE WATCHDOG FROM HAGENBUCH MISSING
; rung 37: ALARM 1-1463 ANALOG OUTPUT FOR ISLAND CONTROL (HAGENBUCH PLC) NOT OK OR PASSIVATED
LD P_On
OUT TR0
ANDNOT I_HAG_BIT_04  ; HAGENBUCH ANALOG OUTPUT NOT OK
SET M_ALARM_1_1463  ; ALARM 1-1463 ANALOG OUTPUT FOR ISLAND CONTROL (HAGENBUCH PLC) NOT OK OR PASSIVATED
LD TR0
AND M_ALARM_1_1463  ; ALARM 1-1463 ANALOG OUTPUT FOR ISLAND CONTROL (HAGENBUCH PLC) NOT OK OR PASSIVATED
OUT LINK_TO_PLC1_ALARM_1_1463  ; LINK TO PLC 1 ALARM 1 1463

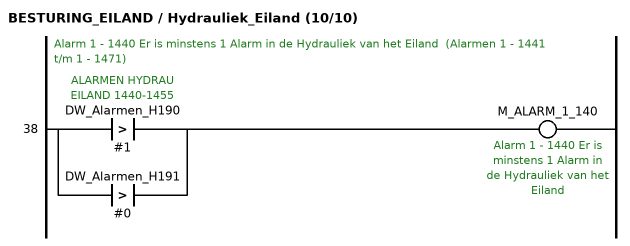
; rung 38: Alarm 1 - 1440 Er is minstens 1 Alarm in de Hydrauliek van het Eiland  (Alarmen 1 - 1441 t/m 1 - 1471)
LD>(320) DW_Alarmen_H190 #1  ; ALARMEN HYDRAU EILAND 1440-1455
OR>(320) DW_Alarmen_H191 #0
OUT M_ALARM_1_140  ; Alarm 1 - 1440 Er is minstens 1 Alarm in de Hydrauliek van het Eiland

### Section Stabilisatie_Eiland

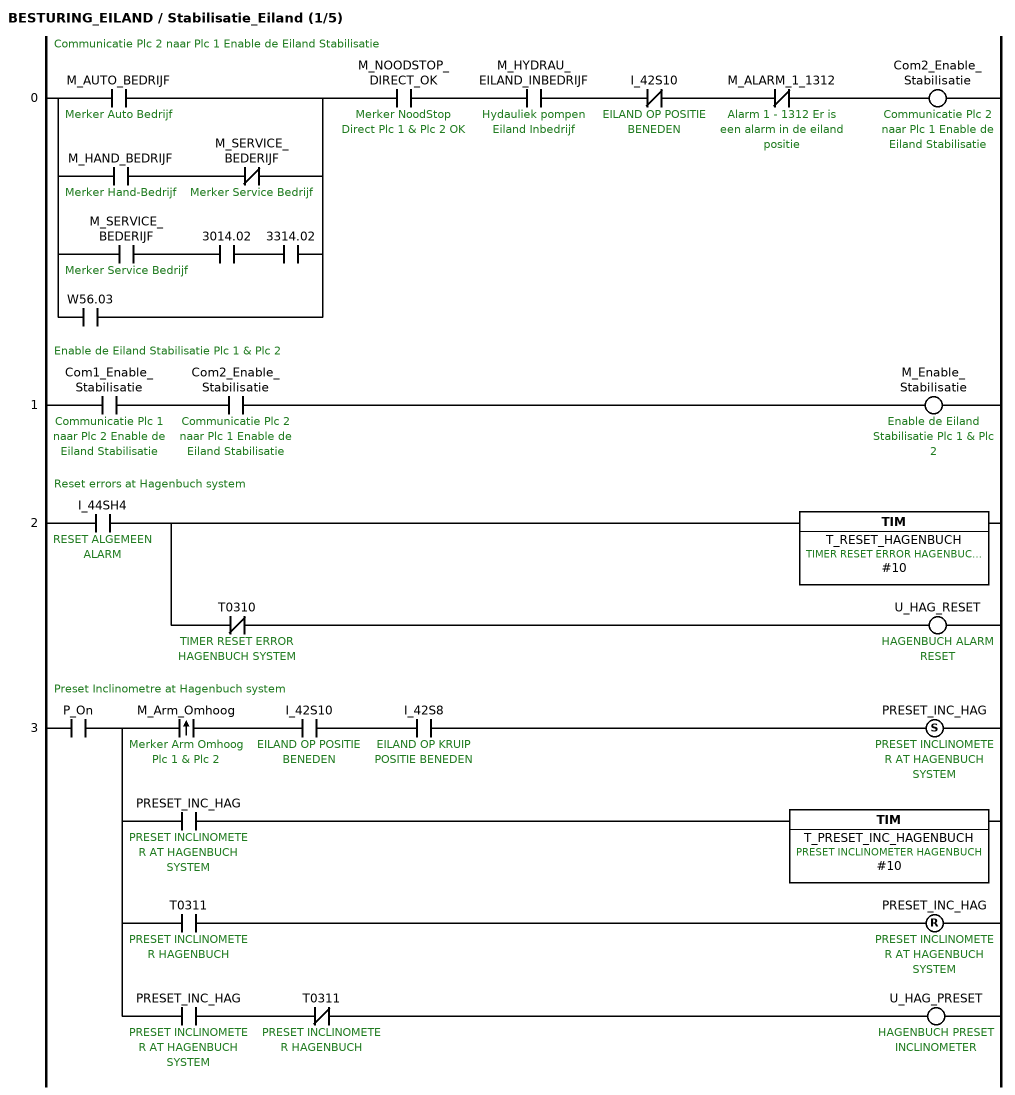
; rung 0: Communicatie Plc 2 naar Plc 1 Enable de Eiland Stabilisatie
LD M_AUTO_BEDRIJF  ; Merker Auto Bedrijf
LD M_HAND_BEDRIJF  ; Merker Hand-Bedrijf
ANDNOT M_SERVICE_BEDERIJF  ; Merker Service Bedrijf
ORLD
LD M_SERVICE_BEDERIJF  ; Merker Service Bedrijf
AND 3014.02
AND 3314.02
ORLD
OR W56.03
AND M_NOODSTOP_DIRECT_OK  ; Merker NoodStop Direct Plc 1 & Plc 2 OK
AND M_HYDRAU_EILAND_INBEDRIJF  ; Hydauliek pompen Eiland Inbedrijf
ANDNOT I_42S10  ; EILAND OP POSITIE BENEDEN
ANDNOT M_ALARM_1_1312  ; Alarm 1 - 1312 Er is een alarm in de eiland positie
OUT Com2_Enable_Stabilisatie  ; Communicatie Plc 2 naar Plc 1 Enable de Eiland Stabilisatie
; rung 1: Enable de Eiland Stabilisatie Plc 1 & Plc 2
LD Com1_Enable_Stabilisatie  ; Communicatie Plc 1 naar Plc 2 Enable de Eiland Stabilisatie
AND Com2_Enable_Stabilisatie  ; Communicatie Plc 2 naar Plc 1 Enable de Eiland Stabilisatie
OUT M_Enable_Stabilisatie  ; Enable de Eiland Stabilisatie Plc 1 & Plc 2
; rung 2: Reset errors at Hagenbuch system
LD I_44SH4  ; RESET ALGEMEEN ALARM
TIM T_RESET_HAGENBUCH #10  ; TIMER RESET ERROR HAGENBUCH SYSTEM
ANDNOT T0310  ; TIMER RESET ERROR HAGENBUCH SYSTEM
OUT U_HAG_RESET  ; HAGENBUCH ALARM RESET
; rung 3: Preset Inclinometre at Hagenbuch system
LD P_On
OUT TR0
@AND M_Arm_Omhoog  ; Merker Arm Omhoog Plc 1 & Plc 2
AND I_42S10  ; EILAND OP POSITIE BENEDEN
AND I_42S8  ; EILAND OP KRUIP POSITIE BENEDEN
SET PRESET_INC_HAG  ; PRESET INCLINOMETER AT HAGENBUCH SYSTEM
LD TR0
AND PRESET_INC_HAG  ; PRESET INCLINOMETER AT HAGENBUCH SYSTEM
TIM T_PRESET_INC_HAGENBUCH #10  ; PRESET INCLINOMETER HAGENBUCH
LD TR0
AND T0311  ; PRESET INCLINOMETER HAGENBUCH
RSET PRESET_INC_HAG  ; PRESET INCLINOMETER AT HAGENBUCH SYSTEM
LD TR0
AND PRESET_INC_HAG  ; PRESET INCLINOMETER AT HAGENBUCH SYSTEM
ANDNOT T0311  ; PRESET INCLINOMETER HAGENBUCH
OUT U_HAG_PRESET  ; HAGENBUCH PRESET INCLINOMETER

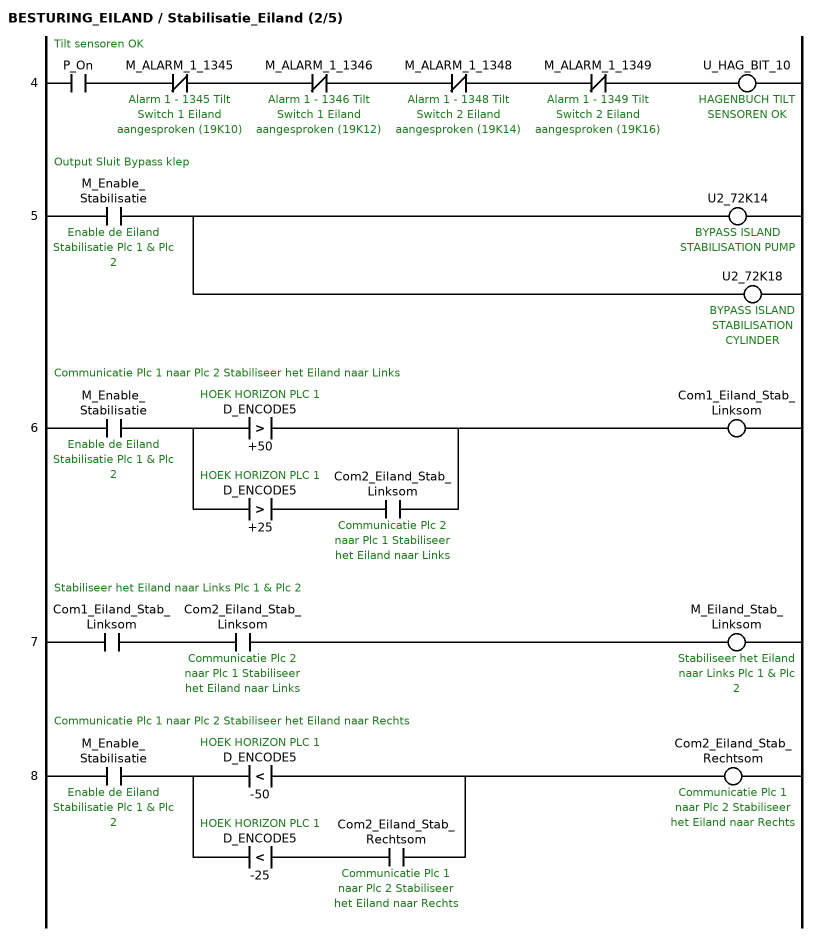
; rung 4: Tilt sensoren OK
LD P_On
ANDNOT M_ALARM_1_1345  ; Alarm 1 - 1345 Tilt Switch 1 Eiland aangesproken (19K10)
ANDNOT M_ALARM_1_1346  ; Alarm 1 - 1346 Tilt Switch 1 Eiland aangesproken (19K12)
ANDNOT M_ALARM_1_1348  ; Alarm 1 - 1348 Tilt Switch 2 Eiland aangesproken (19K14)
ANDNOT M_ALARM_1_1349  ; Alarm 1 - 1349 Tilt Switch 2 Eiland aangesproken (19K16)
OUT U_HAG_BIT_10  ; HAGENBUCH TILT SENSOREN OK
; rung 5: Output Sluit Bypass klep
LD M_Enable_Stabilisatie  ; Enable de Eiland Stabilisatie Plc 1 & Plc 2
OUT U2_72K14  ; BYPASS ISLAND STABILISATION PUMP
OUT U2_72K18  ; BYPASS ISLAND STABILISATION CYLINDER
; rung 6: Communicatie Plc 1 naar Plc 2 Stabiliseer het Eiland naar Links
LD M_Enable_Stabilisatie  ; Enable de Eiland Stabilisatie Plc 1 & Plc 2
LD>S(322) D_ENCODE5 +50  ; HOEK HORIZON PLC 1
LD>S(322) D_ENCODE5 +25  ; HOEK HORIZON PLC 1
AND Com2_Eiland_Stab_Linksom  ; Communicatie Plc 2 naar Plc 1 Stabiliseer het Eiland naar Links
ORLD
ANDLD
OUT Com1_Eiland_Stab_Linksom
; rung 7: Stabiliseer het Eiland naar Links Plc 1 & Plc 2
LD Com1_Eiland_Stab_Linksom
AND Com2_Eiland_Stab_Linksom  ; Communicatie Plc 2 naar Plc 1 Stabiliseer het Eiland naar Links
OUT M_Eiland_Stab_Linksom  ; Stabiliseer het Eiland naar Links Plc 1 & Plc 2
; rung 8: Communicatie Plc 1 naar Plc 2 Stabiliseer het Eiland naar Rechts
LD M_Enable_Stabilisatie  ; Enable de Eiland Stabilisatie Plc 1 & Plc 2
LD<S(312) D_ENCODE5 -50  ; HOEK HORIZON PLC 1
LD<S(312) D_ENCODE5 -25  ; HOEK HORIZON PLC 1
AND Com2_Eiland_Stab_Rechtsom  ; Communicatie Plc 1 naar Plc 2 Stabiliseer het Eiland naar Rechts
ORLD
ANDLD
OUT Com2_Eiland_Stab_Rechtsom  ; Communicatie Plc 1 naar Plc 2 Stabiliseer het Eiland naar Rechts

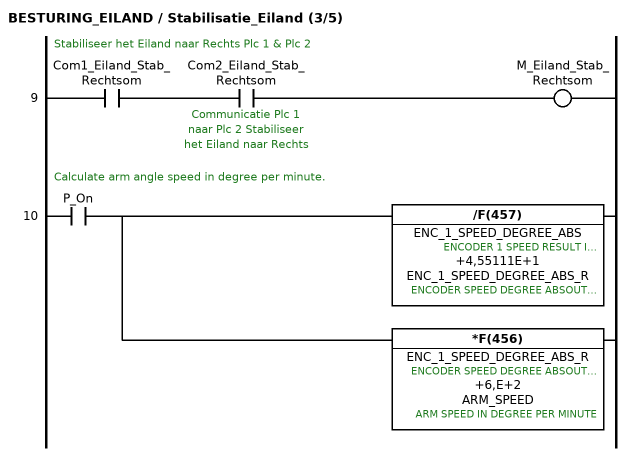
; rung 9: Stabiliseer het Eiland naar Rechts Plc 1 & Plc 2
LD Com1_Eiland_Stab_Rechtsom
AND Com2_Eiland_Stab_Rechtsom  ; Communicatie Plc 1 naar Plc 2 Stabiliseer het Eiland naar Rechts
OUT M_Eiland_Stab_Rechtsom
; rung 10: Calculate arm angle speed in degree per minute.
LD P_On
/F(457) ENC_1_SPEED_DEGREE_ABS +4,55111E+1 ENC_1_SPEED_DEGREE_ABS_R  ; ENCODER 1 SPEED RESULT IN DEGREE ABSOLUTE, ENCODER SPEED DEGREE ABSOUTE REAL
*F(456) ENC_1_SPEED_DEGREE_ABS_R +6,E+2 ARM_SPEED  ; ENCODER SPEED DEGREE ABSOUTE REAL, ARM SPEED IN DEGREE PER MINUTE

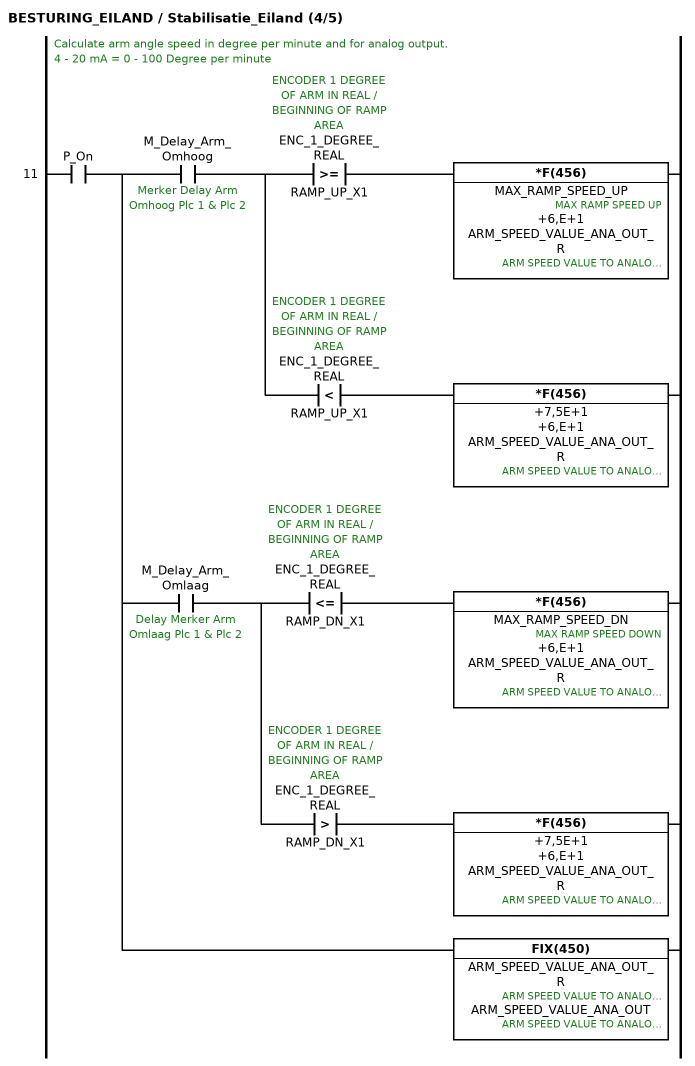
; rung 11: Calculate arm angle speed in degree per minute and for analog output. / 4 - 20 mA = 0 - 100 Degree per minute
LD P_On
OUT TR0
AND M_Delay_Arm_Omhoog  ; Merker Delay Arm Omhoog Plc 1 & Plc 2
OUT TR1
AND>=F(334) ENC_1_DEGREE_REAL RAMP_UP_X1  ; ENCODER 1 DEGREE OF ARM IN REAL, BEGINNING OF RAMP AREA
*F(456) MAX_RAMP_SPEED_UP +6,E+1 ARM_SPEED_VALUE_ANA_OUT_R  ; MAX RAMP SPEED UP, ARM SPEED VALUE TO ANALOG OUTPUT REAL
LD TR1
AND<F(331) ENC_1_DEGREE_REAL RAMP_UP_X1  ; ENCODER 1 DEGREE OF ARM IN REAL, BEGINNING OF RAMP AREA
*F(456) +7,5E+1 +6,E+1 ARM_SPEED_VALUE_ANA_OUT_R  ; ARM SPEED VALUE TO ANALOG OUTPUT REAL
LD TR0
AND M_Delay_Arm_Omlaag  ; Delay Merker Arm Omlaag Plc 1 & Plc 2
OUT TR1
AND<=F(332) ENC_1_DEGREE_REAL RAMP_DN_X1  ; ENCODER 1 DEGREE OF ARM IN REAL, BEGINNING OF RAMP AREA
*F(456) MAX_RAMP_SPEED_DN +6,E+1 ARM_SPEED_VALUE_ANA_OUT_R  ; MAX RAMP SPEED DOWN, ARM SPEED VALUE TO ANALOG OUTPUT REAL
LD TR1
AND>F(333) ENC_1_DEGREE_REAL RAMP_DN_X1  ; ENCODER 1 DEGREE OF ARM IN REAL, BEGINNING OF RAMP AREA
*F(456) +7,5E+1 +6,E+1 ARM_SPEED_VALUE_ANA_OUT_R  ; ARM SPEED VALUE TO ANALOG OUTPUT REAL
LD TR0
FIX(450) ARM_SPEED_VALUE_ANA_OUT_R ARM_SPEED_VALUE_ANA_OUT  ; ARM SPEED VALUE TO ANALOG OUTPUT REAL, ARM SPEED VALUE TO ANALOG OUTPUT

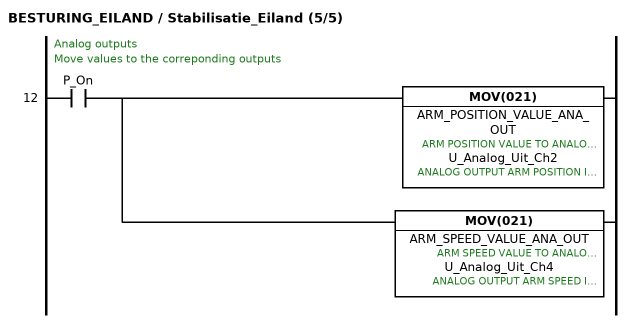
; rung 12: Analog outputs / Move values to the correponding outputs
LD P_On
MOV(021) ARM_POSITION_VALUE_ANA_OUT U_Analog_Uit_Ch2  ; ARM POSITION VALUE TO ANALOG OUTPUT, ANALOG OUTPUT ARM POSITION IN DEGREE
MOV(021) ARM_SPEED_VALUE_ANA_OUT U_Analog_Uit_Ch4  ; ARM SPEED VALUE TO ANALOG OUTPUT, ANALOG OUTPUT ARM SPEED IN DEGREE/MINUTE

### Section Rotatie_Eiland

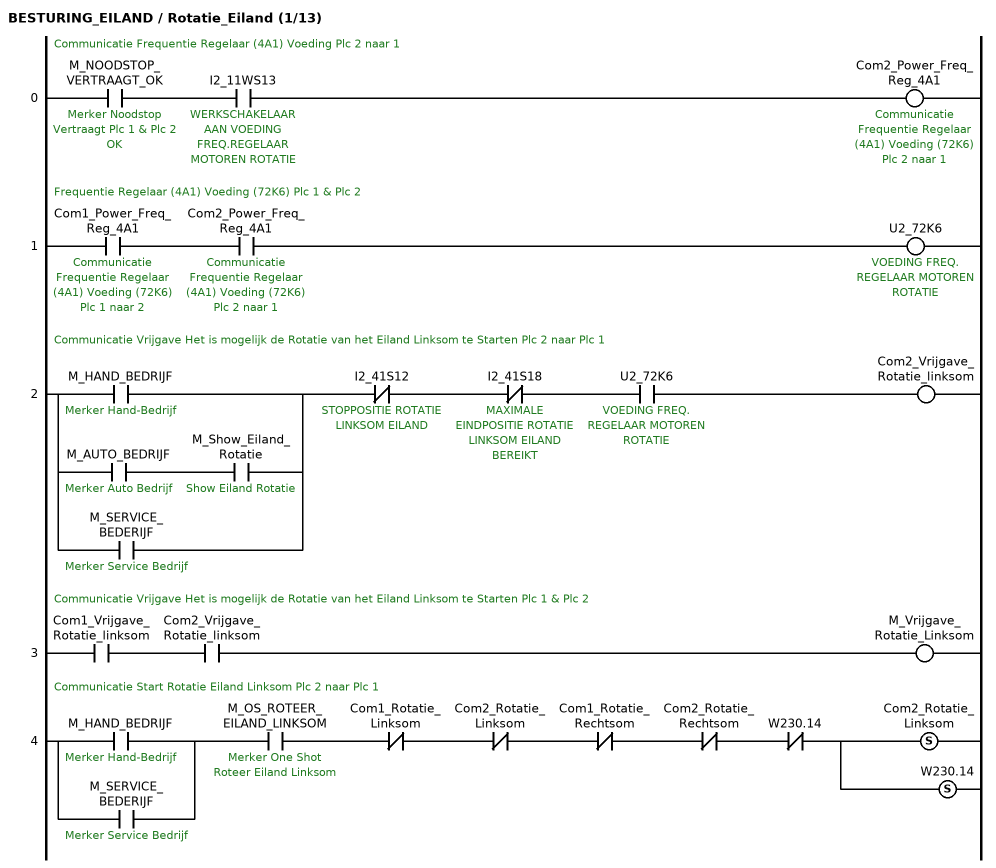
; rung 0: Communicatie Frequentie Regelaar (4A1) Voeding Plc 2 naar 1
LD M_NOODSTOP_VERTRAAGT_OK  ; Merker Noodstop Vertraagt Plc 1 & Plc 2 OK
AND I2_11WS13  ; WERKSCHAKELAAR AAN VOEDING FREQ.REGELAAR MOTOREN ROTATIE
OUT Com2_Power_Freq_Reg_4A1  ; Communicatie Frequentie Regelaar (4A1) Voeding (72K6) Plc 2 naar 1
; rung 1: Frequentie Regelaar (4A1) Voeding (72K6) Plc 1 & Plc 2
LD Com1_Power_Freq_Reg_4A1  ; Communicatie Frequentie Regelaar (4A1) Voeding (72K6) Plc 1 naar 2
AND Com2_Power_Freq_Reg_4A1  ; Communicatie Frequentie Regelaar (4A1) Voeding (72K6) Plc 2 naar 1
OUT U2_72K6  ; VOEDING FREQ.REGELAAR MOTOREN ROTATIE
; rung 2: Communicatie Vrijgave Het is mogelijk de Rotatie van het Eiland Linksom te Starten Plc 2 naar Plc 1
LD M_HAND_BEDRIJF  ; Merker Hand-Bedrijf
LD M_AUTO_BEDRIJF  ; Merker Auto Bedrijf
AND M_Show_Eiland_Rotatie  ; Show Eiland Rotatie
ORLD
OR M_SERVICE_BEDERIJF  ; Merker Service Bedrijf
ANDNOT I2_41S12  ; STOPPOSITIE ROTATIE LINKSOM EILAND
ANDNOT I2_41S18  ; MAXIMALE EINDPOSITIE ROTATIE LINKSOM EILAND BEREIKT
AND U2_72K6  ; VOEDING FREQ.REGELAAR MOTOREN ROTATIE
OUT Com2_Vrijgave_Rotatie_linksom
; rung 3: Communicatie Vrijgave Het is mogelijk de Rotatie van het Eiland Linksom te Starten Plc 1 & Plc 2
LD Com1_Vrijgave_Rotatie_linksom
AND Com2_Vrijgave_Rotatie_linksom
OUT M_Vrijgave_Rotatie_Linksom
; rung 4: Communicatie Start Rotatie Eiland Linksom Plc 2 naar Plc 1
LD M_HAND_BEDRIJF  ; Merker Hand-Bedrijf
OR M_SERVICE_BEDERIJF  ; Merker Service Bedrijf
AND M_OS_ROTEER_EILAND_LINKSOM  ; Merker One Shot Roteer Eiland Linksom
ANDNOT Com1_Rotatie_Linksom
ANDNOT Com2_Rotatie_Linksom
ANDNOT Com1_Rotatie_Rechtsom
ANDNOT Com2_Rotatie_Rechtsom
ANDNOT W230.14
SET Com2_Rotatie_Linksom
SET W230.14

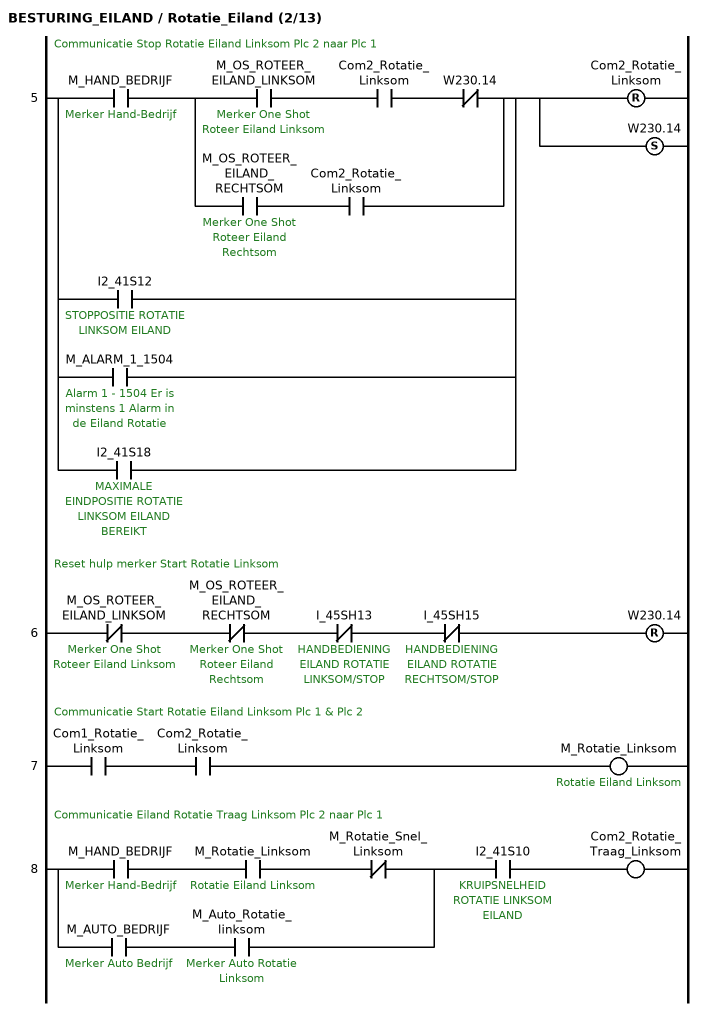
; rung 5: Communicatie Stop Rotatie Eiland Linksom Plc 2 naar Plc 1
LD M_HAND_BEDRIJF  ; Merker Hand-Bedrijf
LD M_OS_ROTEER_EILAND_LINKSOM  ; Merker One Shot Roteer Eiland Linksom
AND Com2_Rotatie_Linksom
ANDNOT W230.14
LD M_OS_ROTEER_EILAND_RECHTSOM  ; Merker One Shot Roteer Eiland Rechtsom
AND Com2_Rotatie_Linksom
ORLD
ANDLD
OR I2_41S12  ; STOPPOSITIE ROTATIE LINKSOM EILAND
OR M_ALARM_1_1504  ; Alarm 1 - 1504 Er is minstens 1 Alarm in de Eiland Rotatie
OR I2_41S18  ; MAXIMALE EINDPOSITIE ROTATIE LINKSOM EILAND BEREIKT
RSET Com2_Rotatie_Linksom
SET W230.14
; rung 6: Reset hulp merker Start Rotatie Linksom
LDNOT M_OS_ROTEER_EILAND_LINKSOM  ; Merker One Shot Roteer Eiland Linksom
ANDNOT M_OS_ROTEER_EILAND_RECHTSOM  ; Merker One Shot Roteer Eiland Rechtsom
ANDNOT I_45SH13  ; HANDBEDIENING EILAND ROTATIE LINKSOM/STOP
ANDNOT I_45SH15  ; HANDBEDIENING EILAND ROTATIE RECHTSOM/STOP
RSET W230.14
; rung 7: Communicatie Start Rotatie Eiland Linksom Plc 1 & Plc 2
LD Com1_Rotatie_Linksom
AND Com2_Rotatie_Linksom
OUT M_Rotatie_Linksom  ; Rotatie Eiland Linksom
; rung 8: Communicatie Eiland Rotatie Traag Linksom Plc 2 naar Plc 1
LD M_HAND_BEDRIJF  ; Merker Hand-Bedrijf
AND M_Rotatie_Linksom  ; Rotatie Eiland Linksom
ANDNOT M_Rotatie_Snel_Linksom
LD M_AUTO_BEDRIJF  ; Merker Auto Bedrijf
AND M_Auto_Rotatie_linksom  ; Merker Auto Rotatie Linksom
ORLD
AND I2_41S10  ; KRUIPSNELHEID ROTATIE LINKSOM EILAND
OUT Com2_Rotatie_Traag_Linksom

